PROGRAM MainProgram
VAR
    counter : INT := 0;
    running : BOOL := FALSE;
END_VAR

IF running THEN
    counter := counter + 1;
    IF counter > 10 THEN
        running := FALSE;
        counter := 0;
    END_IF;
END_IF;

END_PROGRAM

(* stored: Version 1.1.0.1, ProductVersion 3.1.4024.12
   POU MainProgram: Id {a1b2c3d4-e5f6-4a7b-8c9d-0e1f2a3b4c5d}, SpecialFunc None *)
